TYPE ST_VacuumValve :
STRUCT

	//Discrete controls
	i_xSol	 AT%I*	:BOOL;//Solenoid to control the valve( either closed or open)
	
	//Discrete readbacks
	q_xOpnLS  AT%Q*: BOOL;//readback whether open
	q_xClsLS  AT%Q*: BOOL;//readback whether closed
END_STRUCT
END_TYPE

(* stored: Version 1.1.0.1, ProductVersion 3.1.4020.12
   DUT ST_VacuumValve: Id {f7422996-9a0c-4118-9e9f-b51af9eb0c62} *)
